FUNCTION "JsonW_LNK_FixtureSub" : Void
{ S7_Optimized_Access := 'TRUE' }
VERSION : 0.1
   VAR_IN_OUT
      Buf : Array[*] of Byte;   // 출력 버퍼
      Pos : DInt;   // 다음 쓸 절대 인덱스 (< 0 = 오류 유지)
      Val : "LNK_FixtureSub";   // 쓸 값
   END_VAR

   VAR_TEMP
      i0 : DInt;
   END_VAR


BEGIN
	// GENERATED by gr-contract gen-link from "LNK_FixtureSub" sig 16#AFBB75A6 - do not edit
	// wire-spec 2 : 선언 순서, 공백 없음. 버퍼가 모자라면 Pos := LNK_JERR_OVERFLOW (끈끈한 오류, 호출자가 끝에 한 번 확인)
	"Json_WRaw"(Buf := #Buf, Pos := #Pos, Lit := '{"Id":');
	"Json_WUInt"(Buf := #Buf, Pos := #Pos, Val := #Val.Id);
	"Json_WRaw"(Buf := #Buf, Pos := #Pos, Lit := ',"Name":');
	"Json_WStr"(Buf := #Buf, Pos := #Pos, Val := #Val.Name);
	"Json_WRaw"(Buf := #Buf, Pos := #Pos, Lit := ',"On":');
	"Json_WBool"(Buf := #Buf, Pos := #Pos, Val := #Val.On);
	"Json_WRaw"(Buf := #Buf, Pos := #Pos, Lit := ',"Pos":[');
	FOR #i0 := 1 TO 4 DO   // "X".."G"
	  IF #i0 > 1 THEN
	    "Json_WComma"(Buf := #Buf, Pos := #Pos);
	  END_IF;
	  "Json_WReal"(Buf := #Buf, Pos := #Pos, Val := #Val.Pos[#i0]);
	END_FOR;
	"Json_WRaw"(Buf := #Buf, Pos := #Pos, Lit := ']}');
END_FUNCTION
